{attribute 'qualified_only'}
{attribute 'strict'}
{attribute 'to_string'}
TYPE E_Reaction :
(
	Complete 			:= 300,
	StopCycle   		:= 400, 
    Stop  	 			:= 500,
	Abort    			:= 600
 );	
END_TYPE

(* stored: Version 1.1.0.1
   DUT E_Reaction: Id {d2151b9b-4367-42a7-936d-7f67fb250d47} *)
